// TIA Portal V16 export
// export: Created 2020-03-21T19:11:08.7154816Z, ExportSetting None, DisplayName Totally Integrated Automation Portal, DisplayVersion V16, DisplayName TIA Portal Version Control Interface, DisplayVersion V16, DisplayName TIA Portal Openness, DisplayVersion V16, DisplayName SINAMICS Startdrive Advanced, DisplayVersion V16, DisplayName SINAMICS Startdrive G130, G150, S120, S150, SINAMICS MV, S210, DisplayVersion V16, DisplayName SINAMICS Startdrive G110M, G120, G120C, G120D, G120P, DisplayVersion V16, DisplayName STEP 7 Professional, DisplayVersion V16, DisplayName STEP 7 Safety, DisplayVersion V16, DisplayName WinCC Advanced, DisplayVersion V16
FUNCTION "Block_2" : Void   // FC1, LAD
TITLE = Block Title
{ S7_Optimized_Access := 'TRUE' }
// Block Kommentar 1
// stored: SetENOAutomatically false
BEGIN

REGION Network 1: Netzwerk 1
   // Netzwerk Kommentar 1
END_REGION
END_FUNCTION
